// TwinCAT 3 PLC project TcLog
// Title: TcLog
// Company: TcLog
// ProjectVersion: 0.5.0
// ProgramVersion: 3.1.4022.7
// libraries:
//   Tc2_Standard, * (Beckhoff Automation GmbH)
//   Tc2_System, * (Beckhoff Automation GmbH)
//   Tc2_Utilities, * (Beckhoff Automation GmbH)
//   Tc3_Module, * (Beckhoff Automation GmbH)
//   TcExt, * (TcExt)
//   TcUnit, * (www.tcunit.org)
// project tree:
//   Event/ CyclicEventDetection.TcPOU, EventMessageHMI.TcDUT, ST_CyclicMessageDetection.TcDUT, Event.TcPOU, EventLevel.TcDUT, EventMessage.TcDUT, EventRunner.TcPOU, ST_CyclicEventDetection.TcDUT
//   / GlobalTextList.TcGTLO, SymbolsPool.TcIPO (not stored), Visualization Manager.TcVMO (not stored)
//   GVL/ GVL.TcGVL, Properties.TcGVL
//   Logger/ ADSLogger.TcPOU, EventLogger.TcIO, CSVLogger.TcPOU, MemoryLogger.TcPOU, AlarmViewLogger.TcPOU
//   Tests/Event/ EventTestsystem.TcDUT, MultipleEventTestsystem.TcDUT, TestEvent.TcPOU
//   Tests/Logger/ ADSLoggerTestsystem.TcDUT, CSVLoggerTestsystem.TcDUT, TestADSLogger.TcPOU, TestCSVLogger.TcPOU
//   Tests/ PlcTask.TcTTO, TEST_MAIN.TcPOU, TEST_STRING_CYCLE_TIME.TcPOU
//   Tests/Utils/ TestUtils.TcPOU
//   Utils/ FB_FrameFifo.TcPOU, LString.TcPOU, put_new_data_at_start.TcPOU, remove_field_from_array.TcPOU, TIMESTRUCT_TO_DATESTR.TcPOU, TIMESTRUCT_TO_TIMESTR.TcPOU, TO_LSTRING.TcPOU
//   Visu/ AlarmViewMulti.TcVIS, AlarmViewSingle.TcVIS, AlarmViewSingleWithReset.TcVIS
// real-time tasks:
//   TASK PlcTask: cycle T#10ms, priority 20, ADS port 350

CONFIGURATION TcLog
    RESOURCE PLC ON TwinCAT3
        TASK PlcTask(INTERVAL := T#10ms, PRIORITY := 20);
    END_RESOURCE
END_CONFIGURATION

// ---- Event/EventMessageHMI.TcDUT
TYPE EventMessageHMI :
STRUCT
  id: INT;
  timestamp: STRING;
  path: STRING;
  message: STRING;
  level: EventLevel;
END_STRUCT
END_TYPE

// ---- Event/ST_CyclicMessageDetection.TcDUT
TYPE ST_CyclicMessageDetection :
STRUCT
  ev: EventMessage;
  message_submitted: BOOL;
END_STRUCT
END_TYPE

// ---- Event/EventLevel.TcDUT
{attribute 'qualified_only'}
{attribute 'strict'}
{attribute 'to_string'}
TYPE EventLevel :
(
  NONE := 0,
  DEBUG := 1,
	INFO := 2,
  WARNING := 3,
  ERROR := 4,
  ALARM := 5
) BYTE := NONE;
END_TYPE

// ---- Event/EventMessage.TcDUT
TYPE EventMessage :
STRUCT
  id: INT;
  path: LString;
  message: LString;
  level: EventLevel;
  cleared: BOOL;
END_STRUCT
END_TYPE

// ---- Event/ST_CyclicEventDetection.TcDUT
TYPE ST_CyclicEventDetection :
STRUCT
  id: INT;
  submitted_in_last_invocation: BIT;
END_STRUCT
END_TYPE

// ---- Tests/Event/EventTestsystem.TcDUT
TYPE EventTestsystem :
STRUCT
  logging: EventRunner;
  event: Event := (logging:=logging);
END_STRUCT
END_TYPE

// ---- Tests/Event/MultipleEventTestsystem.TcDUT
TYPE MultipleEventTestsystem :
STRUCT
  logging: EventRunner;
  event1: Event := (logging:=logging);
  event2: Event := (logging:=logging);
  event3: Event := (logging:=logging);
END_STRUCT
END_TYPE

// ---- Tests/Logger/ADSLoggerTestsystem.TcDUT
TYPE ADSLoggerTestsystem :
STRUCT
  logging: EventRunner;
  event: Event := (logging:=logging);
  logger: ADSLogger := (disable_ads_output := TRUE);
END_STRUCT
END_TYPE

// ---- Tests/Logger/CSVLoggerTestsystem.TcDUT
TYPE CSVLoggerTestsystem :
STRUCT
  logging: EventRunner;
  event: Event := (logging:=logging);
  logger: CSVLogger;
END_STRUCT
END_TYPE

// ---- GVL/GVL.TcGVL
VAR_GLOBAL
  logging: EventRunner;
END_VAR
VAR_GLOBAL CONSTANT
  EXCLUDE_ID: INT := 0;
  // Index zero should not be visible
  IMAGE_ID: ARRAY[0..5] OF STRING(20) := ['SymbolsPool.info', 'SymbolsPool.info', 'SymbolsPool.info', 'SymbolsPool.warning', 'SymbolsPool.error', 'SymbolsPool.alarm'];
END_VAR

// ---- GVL/Properties.TcGVL
{attribute 'qualified_only'}
VAR_GLOBAL CONSTANT
  NUM_EVENTS: INT := 500;
  NUM_CONCURRENT_ALARMS: INT := 10;
  NUM_LOGGER: INT := 5;
  NUM_CYCLIC_DETECTION_MESSAGES: INT := 10;
  CSV_BUFFER_SIZE: UDINT := 2000;
  MEMORY_LOGGER_NUM_EVENTS_HISTORY: INT := 100;
  MEMORY_LOGGER_NUM_EVENTS_HMI: INT := 30;
  ALARM_VIEW_NUM_EVENTS: INT := 20;
END_VAR

// ---- Logger/EventLogger.TcIO
INTERFACE EventLogger

METHOD clear_event_message
VAR_INPUT
  id: INT;
END_VAR
END_METHOD

PROPERTY PUBLIC level : EventLevel
GET
END_GET
SET
END_SET
END_PROPERTY

METHOD run
VAR_INPUT
  act_time: TIMESTRUCT;
END_VAR
END_METHOD

METHOD PUBLIC submit_event_message
VAR_IN_OUT
  ev: EventMessage;
END_VAR
END_METHOD

END_INTERFACE

// ---- Event/EventRunner.TcPOU
{attribute 'reflection'}
FUNCTION_BLOCK EventRunner
VAR_INPUT
END_VAR
VAR_OUTPUT
END_VAR
VAR
  {attribute 'instance-path'}
  {attribute 'noinit'}
  path_str: STRING(255);
  path: LString;
  event_id_counter: INT;
  localtime: FB_LocalSystemTime := (bEnable:=TRUE);
  actSystemTime: TIMESTRUCT;
  event_logger: ARRAY[1..Properties.NUM_LOGGER] OF EventLogger;
  active_alarms: ARRAY[1..Properties.NUM_CONCURRENT_ALARMS] OF EventMessage;
  detection: CyclicEventDetection;
  logger_counter: INT;
  format_str: FB_FormatString;
  _parameter: T_Arg;
  
  submit_event_message_counter: INT;
  max_submit_event_message_counter: INT;
END_VAR

(* 
der runner wird am ende des sps programms ausgefuehrt
- im programm werden pro meldung event-instanzen erstellt. diese registrieren sich selbst. die richtige id wird der pfad zur instanzvariable sein
- im runner wird zudem das datum immer aktualisiert
*)

PROPERTY PRIVATE act_time : TIMESTRUCT
GET
IF time_valid THEN
  act_time := localtime.systemTime;
END_IF
END_GET
END_PROPERTY

METHOD PUBLIC add_logger
VAR_INPUT
  logger: EventLogger;
END_VAR
IF logger_counter < Properties.NUM_LOGGER AND ADR(logger) <> 0 AND NOT logger_exist(logger) THEN
  inc_logger_counter();
  event_logger[logger_counter] := logger;
END_IF
END_METHOD

METHOD INTERNAL alarm_raised : BOOL
VAR_INPUT
  id: INT;
END_VAR
VAR
  i: INT;
END_VAR
alarm_raised := get_alarm_index(id:=id) > 0;
END_METHOD

METHOD PUBLIC clear
VAR_INPUT
  id: INT;
END_VAR
VAR
  i: INT;
END_VAR
FOR i:=1 TO Properties.NUM_LOGGER DO
  IF event_logger[i] <> 0 THEN
    event_logger[i].clear_event_message(id);
	END_IF
END_FOR
END_METHOD

METHOD INTERNAL clear_alarm
VAR_INPUT
  id: INT;
END_VAR
VAR
  index: INT;
  filldata: EventMessage;
END_VAR
IF alarm_raised(id:=id) THEN
  index := get_alarm_index(id:=id);
  active_alarms[index].cleared := TRUE;
  
  submit_event_message_to_logger(active_alarms[index]);
  
  remove_field_from_array(
    index_to_remove:=index,
    size_filldata:=SIZEOF(filldata),
    adr_filldata:=ADR(filldata),
    size_memory_buffer:=SIZEOF(active_alarms),
    adr_memory_buffer:=ADR(active_alarms));
END_IF
END_METHOD

METHOD PRIVATE create_event_message
VAR_INPUT
  id: INT;
  level: EventLevel;
  cleared: BOOL;
END_VAR
VAR_IN_OUT
  ev: EventMessage;
  path: LString;
  message: LString;
END_VAR
VAR
  undefined_time: TIMESTRUCT;
  num_dots: INT;
  i: INT;
  offset: INT;
END_VAR
ev.id := id;
ev.path := path;
ev.message := message;
ev.level := level;
ev.cleared := cleared;
END_METHOD

METHOD PUBLIC error
VAR_INPUT
  message: STRING(255);
END_VAR
VAR_INST
  message_lstr: LString;
END_VAR
message_lstr := TO_LSTRING(message);
submit_message(
  message:=message_lstr,
  level:=EventLevel.ERROR);
END_METHOD

METHOD PUBLIC error_if_true
VAR_INPUT
  value: BOOL;
  message: STRING(255);
END_VAR
IF value THEN
  error(message);
END_IF
END_METHOD

METHOD FB_init : BOOL
VAR_INPUT
	bInitRetains : BOOL; // if TRUE, the retain variables are initialized (warm start / cold start)
	bInCopyCode : BOOL;  // if TRUE, the instance afterwards gets moved into the copy code (online change)
END_VAR
path.str := path_str;
END_METHOD

METHOD INTERNAL generate_event_id : INT
VAR_INPUT
END_VAR
inc_event_id_counter();
generate_event_id := event_id_counter;
END_METHOD

METHOD PRIVATE get_alarm_index : INT
VAR_INPUT
  id: INT;
END_VAR
VAR
  i: INT;
END_VAR
get_alarm_index := 0;
FOR i:=1 TO Properties.NUM_CONCURRENT_ALARMS DO
  IF active_alarms[i].id = id AND NOT active_alarms[i].cleared THEN
    get_alarm_index := i;
    EXIT;
	END_IF
END_FOR
END_METHOD

METHOD PRIVATE inc_event_id_counter
VAR_INPUT
END_VAR
event_id_counter := LIMIT(1, event_id_counter + 1, Properties.NUM_EVENTS);
END_METHOD

METHOD PRIVATE inc_logger_counter
VAR_INPUT
END_VAR
logger_counter := LIMIT(1, logger_counter + 1, Properties.NUM_LOGGER);
END_METHOD

METHOD PUBLIC info
VAR_INPUT
  message: STRING(255);
END_VAR
VAR_INST
  message_lstr: LString;
END_VAR
message_lstr := TO_LSTRING(message);
submit_message(
  message:=message_lstr,
  level:=EventLevel.INFO);
END_METHOD

METHOD PUBLIC info_if_true
VAR_INPUT
  value: BOOL;
  message: STRING(255);
END_VAR
IF value THEN
  info(message);
END_IF
END_METHOD

METHOD PRIVATE logger_exist : BOOL
VAR_INPUT
  logger: EventLogger;
END_VAR
VAR
  i: INT;
END_VAR
logger_exist := FALSE;
FOR i:=1 TO Properties.NUM_LOGGER DO
  IF event_logger[i] = logger THEN
    logger_exist := TRUE;
    EXIT;
	END_IF
END_FOR
END_METHOD

PROPERTY PUBLIC parameter : T_Arg
GET
parameter := _parameter;
END_GET
SET
_parameter := parameter;
END_SET
END_PROPERTY

METHOD PUBLIC reset_events_and_messages
VAR_INPUT
END_VAR
detection.reset_events();
detection.reset_messages();
END_METHOD

METHOD PUBLIC run
VAR_INPUT
END_VAR
VAR
  read_done: BOOL;
  error_id: UDINT;
END_VAR
localtime();
run_logger();
detection.cyclic_call();
submit_event_message_counter := 0;
END_METHOD

METHOD PRIVATE run_logger
VAR_INPUT
END_VAR
VAR
  i: INT;
END_VAR
FOR i:=1 TO Properties.NUM_LOGGER DO
  IF event_logger[i] <> 0 THEN
    event_logger[i].run(act_time:=act_time);
	END_IF
END_FOR
END_METHOD

METHOD PUBLIC submit_event
VAR_INPUT
  id: INT;
  level: EventLevel;
  cleared: BOOL;
END_VAR
VAR_IN_OUT
  path: LString;
  message: LString;
END_VAR
VAR
  temp_message: STRING(255);
END_VAR
VAR_INST
  ev: EventMessage;
  event_index: INT;
  message_index: INT;
  formatted_message: LString;
END_VAR
IF alarm_raised(id:=id) THEN
  RETURN;
END_IF

event_index := detection.get_event_index(id);
IF event_index = 0 THEN
  detection.add_event(id);
  IF _parameter.cbLen > 0 THEN
    format_str(
      sFormat:=message.str,
      arg1:=parameter,
      sOut=>temp_message);
    formatted_message.str := temp_message;
  ELSE
    formatted_message := message;
  END_IF
  ev.id := id;
  ev.path := path;
  ev.message := formatted_message;
  ev.level := level;
  ev.cleared := cleared;
  ev.path.remove_left_including_char('.', 2);
  submit_event_message_to_logger(ev);
  
  IF NOT cleared THEN
    put_new_data_at_start(SIZEOF(ev), ADR(ev), SIZEOF(active_alarms), ADR(active_alarms));
  END_IF
ELSE
  detection.reactivate_event(event_index);
END_IF
END_METHOD

METHOD PRIVATE submit_event_message_to_logger
VAR_IN_OUT
  ev: EventMessage;
END_VAR
VAR
  i: INT;
END_VAR
FOR i:=1 TO Properties.NUM_LOGGER DO
  IF event_logger[i] <> 0 THEN
    event_logger[i].submit_event_message(ev);
	END_IF
END_FOR
END_METHOD

METHOD PRIVATE submit_message
VAR_INPUT
  level: EventLevel;
END_VAR
VAR_IN_OUT
  message: LString;
END_VAR
VAR
  temp_message: STRING(255);
END_VAR
VAR_INST
  ev: EventMessage;
  event_index: INT;
  message_index: INT;
  formatted_message: LString;
END_VAR
IF _parameter.cbLen > 0 THEN
  format_str(
    sFormat:=message.str,
    arg1:=parameter,
    sOut=>temp_message);
  formatted_message.str := temp_message;
ELSE
  formatted_message := message;
END_IF
create_event_message(
    ev:=ev,
    id:=GVL.EXCLUDE_ID,
    path:=path,
    message:=formatted_message,
    level:=level,
    cleared:=TRUE);
message_index := detection.get_message_index(ev);
IF message_index = 0 THEN
  ev.path.remove_left_including_char('.', 2);
  detection.add_message(ev);
  
  submit_event_message_to_logger(ev);
ELSE
  detection.reactivate_message(message_index);
END_IF
END_METHOD

PROPERTY PUBLIC time_valid : BOOL
GET
time_valid := localtime.bValid;
END_GET
END_PROPERTY

METHOD PRIVATE timestruct_equal : BOOL
VAR_INPUT
  timestruct_1: TIMESTRUCT;
  timestruct_2: TIMESTRUCT;
END_VAR
timestruct_equal := timestruct_1.wDay = timestruct_2.wDay;
timestruct_equal := timestruct_equal AND timestruct_1.wDayOfWeek = timestruct_2.wDayOfWeek;
timestruct_equal := timestruct_equal AND timestruct_1.wHour = timestruct_2.wHour;
timestruct_equal := timestruct_equal AND timestruct_1.wMilliseconds = timestruct_2.wMilliseconds;
timestruct_equal := timestruct_equal AND timestruct_1.wMinute = timestruct_2.wMinute;
END_METHOD

METHOD PUBLIC warning
VAR_INPUT
  message: STRING(255);
END_VAR
VAR_INST
  message_lstr: LString;
END_VAR
message_lstr := TO_LSTRING(message);
submit_message(
  message:=message_lstr,
  level:=EventLevel.WARNING);
END_METHOD

METHOD PUBLIC warning_if_true
VAR_INPUT
  value: BOOL;
  message: STRING(255);
END_VAR
IF value THEN
  warning(message);
END_IF
END_METHOD

END_FUNCTION_BLOCK

// ---- Utils/LString.TcPOU
FUNCTION_BLOCK LString
VAR_INPUT
END_VAR
VAR_OUTPUT
END_VAR
VAR
  _str: STRING(255);
  _length: INT;
END_VAR

METHOD PUBLIC append
VAR_IN_OUT
  lstr: LString; 
END_VAR
MEMMOVE(
  destAddr:=ADR(_str)+TO_DWORD(length),
  srcAddr:=ADR(lstr._str),
  n:=TO_UDINT(lstr.length+1));
length := length + lstr.length;
END_METHOD

METHOD PUBLIC append_str
VAR_INPUT
  str: STRING(255);
END_VAR
VAR
  length: INT;
END_VAR
length := LEN(str);
MEMMOVE(
  destAddr:=ADR(_str)+TO_DWORD(THIS^.length),
  srcAddr:=ADR(str),
  n:=TO_UDINT(length+1));
THIS^.length := THIS^.length + length;
END_METHOD

PROPERTY PUBLIC length : INT
GET
length := _length;
END_GET
SET // PRIVATE
_length := length;
END_SET
END_PROPERTY

METHOD PUBLIC remove_left_including_char
VAR_INPUT
  char: STRING(1);
  number: INT;
END_VAR
VAR
  act_number: INT;
  offset: INT;
  i: INT;
END_VAR
WHILE _str[i] <> 0 DO
  IF act_number < number THEN
    IF _str[i] = char[0] THEN
      act_number := act_number + 1;
    END_IF
  ELSE
    EXIT;
	END_IF
  i := i + 1;
END_WHILE
MEMMOVE(
  destAddr:=ADR(_str),
  srcAddr:=ADR(_str)+TO_DWORD(i),
  n:=TO_UDINT(length-i));
length := length - i;
_str[length] := 0;
END_METHOD

PROPERTY PUBLIC str : STRING(255)
GET
str := _str;
END_GET
SET
_str := str;
length := LEN(str);
END_SET
END_PROPERTY

END_FUNCTION_BLOCK

// ---- Event/CyclicEventDetection.TcPOU
FUNCTION_BLOCK CyclicEventDetection
VAR_INPUT
END_VAR
VAR_OUTPUT
END_VAR
VAR
  message_counter: INT;
  event_counter: INT;
  messages: ARRAY[1..Properties.NUM_CYCLIC_DETECTION_MESSAGES] OF ST_CyclicMessageDetection;
  events: ARRAY[1..Properties.NUM_EVENTS] OF ST_CyclicEventDetection;
END_VAR

METHOD PRIVATE activate_event
VAR_INPUT
  index: INT;
END_VAR
events[index].submitted_in_last_invocation := TRUE;
END_METHOD

METHOD PRIVATE activate_message
VAR_INPUT
  index: INT;
END_VAR
messages[index].message_submitted := TRUE;
END_METHOD

METHOD PUBLIC add_event
VAR_INPUT
  id: INT;
END_VAR
VAR
  event_index: INT;
END_VAR
inc_event_counter();
events[event_counter].id := id;
activate_event(event_counter);
END_METHOD

METHOD PUBLIC add_message
VAR_INPUT
  ev: EventMessage;
END_VAR
VAR
  event_index: INT;
END_VAR
IF NOT max_number_events_reached() THEN
  inc_message_counter();
  messages[message_counter].ev := ev;
  activate_message(message_counter);
END_IF
END_METHOD

METHOD PUBLIC cyclic_call
VAR_INPUT
END_VAR
remove_deactivated_events();
remove_deactivated_messages();
reset_events();
reset_messages();
END_METHOD

METHOD PRIVATE dec_event_counter
VAR_INPUT
END_VAR
event_counter := LIMIT(0, event_counter - 1, Properties.NUM_EVENTS);
END_METHOD

METHOD PRIVATE dec_message_counter
VAR_INPUT
END_VAR
message_counter := LIMIT(0, message_counter - 1, Properties.NUM_CYCLIC_DETECTION_MESSAGES);
END_METHOD

METHOD PRIVATE event_id_valid : BOOL
VAR_INPUT
  id: INT;
END_VAR
event_id_valid := (1 <= id) AND (id <= Properties.NUM_EVENTS);
END_METHOD

METHOD PUBLIC event_was_called_in_last_invocation : BOOL
VAR_INPUT
  id: INT;
END_VAR
VAR
  i: INT;
END_VAR
FOR i:=1 TO event_counter DO
  IF events[i].id = id THEN
    event_was_called_in_last_invocation := TRUE;
    EXIT;
	END_IF
END_FOR
END_METHOD

METHOD PUBLIC get_event_index : INT
VAR_INPUT
  id: INT;
END_VAR
VAR
  i: INT;
END_VAR
FOR i:=1 TO event_counter DO
  IF events[i].id = id THEN
    get_event_index := i;
    EXIT;
  END_IF
END_FOR
END_METHOD

METHOD get_message_index : INT
VAR_IN_OUT
  ev: EventMessage;
END_VAR
VAR
  i: INT;
END_VAR
FOR i:=1 TO message_counter DO
  IF messages[i].ev.message.str = ev.message.str THEN
    get_message_index := i;
    EXIT;
  END_IF
END_FOR
END_METHOD

METHOD PRIVATE inc_event_counter
VAR_INPUT
END_VAR
event_counter := LIMIT(1, event_counter + 1, Properties.NUM_EVENTS);
END_METHOD

METHOD PRIVATE inc_message_counter
VAR_INPUT
END_VAR
message_counter := LIMIT(1, message_counter + 1, Properties.NUM_CYCLIC_DETECTION_MESSAGES);
END_METHOD

METHOD PRIVATE max_number_events_reached : BOOL
VAR_INPUT
END_VAR
max_number_events_reached := message_counter >= Properties.NUM_CYCLIC_DETECTION_MESSAGES;
END_METHOD

METHOD PRIVATE message_index_valid : BOOL
VAR_INPUT
  index: INT;
END_VAR
message_index_valid := (1 <= index) AND (index <= Properties.NUM_CYCLIC_DETECTION_MESSAGES);
END_METHOD

METHOD PUBLIC reactivate_event
VAR_INPUT
  index: INT;
END_VAR
IF event_id_valid(index) THEN
  activate_event(index);
END_IF
END_METHOD

METHOD PUBLIC reactivate_message
VAR_INPUT
  index: INT;
END_VAR
IF event_id_valid(index) THEN
  activate_message(index);
END_IF
END_METHOD

METHOD PRIVATE remove_deactivated_events
VAR_INPUT
END_VAR
VAR
  i: INT;
  filldata: ST_CyclicEventDetection;
END_VAR
FOR i:=1 TO event_counter DO
  IF NOT events[i].submitted_in_last_invocation THEN
    remove_field_from_array(
      index_to_remove:=i,
      size_filldata:=SIZEOF(filldata),
      adr_filldata:=ADR(filldata),
      size_memory_buffer:=SIZEOF(events),
      adr_memory_buffer:=ADR(events)
    );
    dec_event_counter();
    i := i - 1;
	END_IF
END_FOR
END_METHOD

METHOD PRIVATE remove_deactivated_messages
VAR_INPUT
END_VAR
VAR
  i: INT;
  filldata: ST_CyclicMessageDetection;
END_VAR
FOR i:=1 TO message_counter DO
  IF NOT messages[i].message_submitted THEN
    remove_field_from_array(
      index_to_remove:=i,
      size_filldata:=SIZEOF(filldata),
      adr_filldata:=ADR(filldata),
      size_memory_buffer:=SIZEOF(messages),
      adr_memory_buffer:=ADR(messages)
    );
    dec_message_counter();
    i := i - 1;
	END_IF
END_FOR
END_METHOD

METHOD PRIVATE reset_event
VAR_INPUT
  index: INT;
END_VAR
events[index].submitted_in_last_invocation := FALSE;
END_METHOD

METHOD PUBLIC reset_events
VAR_INPUT
END_VAR
VAR
  i: INT;
END_VAR
FOR i:=1 TO event_counter DO
  reset_event(i);
END_FOR
END_METHOD

METHOD PRIVATE reset_message
VAR_INPUT
  index: INT;
END_VAR
messages[index].message_submitted := FALSE;
END_METHOD

METHOD PUBLIC reset_messages
VAR_INPUT
END_VAR
VAR
  i: INT;
END_VAR
FOR i:=1 TO message_counter DO
  reset_message(i);
END_FOR
END_METHOD

END_FUNCTION_BLOCK

// ---- Utils/remove_field_from_array.TcPOU
FUNCTION remove_field_from_array : BOOL
VAR_INPUT
  index_to_remove: INT; // array index must start with 1
  size_filldata: UDINT;
  adr_filldata: POINTER TO BYTE; 
  size_memory_buffer: UDINT;
  adr_memory_buffer : POINTER TO BYTE;
END_VAR
VAR
END_VAR

IF index_to_remove < 1 THEN
  RETURN;
END_IF

(*
example:
size_memory_buffer = 20
size_filldata = 1
index_to_remove = 1
adr_memory_buffer = 100
---------------------------------
size_new_data = 20 - 1 = 19
adr_new_data = 100 + 1 = 101


size_memory_buffer = 20 - 1 = 19
adr_memory_buffer = 100 + 0 = 100
*)

FW_MemMove(
  pDest := adr_memory_buffer + size_filldata*TO_UDINT((index_to_remove-1)),
  pSrc := adr_memory_buffer + size_filldata*TO_UDINT(index_to_remove),
  cbLen := size_memory_buffer - size_filldata*TO_UDINT(index_to_remove));
FW_MemMove(
  pDest := adr_memory_buffer + (size_memory_buffer - size_filldata),
  pSrc := adr_filldata,
  cbLen := size_filldata);

END_FUNCTION

// ---- Utils/TO_LSTRING.TcPOU
FUNCTION TO_LSTRING : LSTRING
VAR_INPUT
  str: STRING(255);
END_VAR
VAR
END_VAR

TO_LSTRING.str := str;

END_FUNCTION

// ---- Utils/put_new_data_at_start.TcPOU
FUNCTION put_new_data_at_start: BOOL
VAR_INPUT
  size_new_data: UDINT;
  adr_new_data: POINTER TO BYTE;

  size_memory_buffer: UDINT;
  adr_memory_buffer : POINTER TO BYTE;
END_VAR

FW_MemMove(
  pDest := adr_memory_buffer + size_new_data,
  pSrc := adr_memory_buffer,
  cbLen := size_memory_buffer - size_new_data);
FW_MemMove(
  pDest := adr_memory_buffer,
  pSrc := adr_new_data,
  cbLen := size_new_data);

END_FUNCTION

// ---- Event/Event.TcPOU
{attribute 'reflection'}
FUNCTION_BLOCK Event
VAR_INPUT
END_VAR
VAR_OUTPUT
END_VAR
VAR
  _logging: REFERENCE TO EventRunner;
  {attribute 'instance-path'}
  {attribute 'noinit'}
  path_str: STRING(255);
  path: LString;
  id: INT;
  _message: LString;
  _parameter: T_Arg;
  ev: EventMessage;
END_VAR

METHOD PUBLIC alarm
VAR_INPUT
END_VAR
submit(level:=EventLevel.ALARM);
END_METHOD

METHOD alarm_if_true
VAR_INPUT
    value: BOOL;
END_VAR
IF value THEN
  alarm();
ELSE
  clear_alarm();
END_IF
END_METHOD

PROPERTY PUBLIC alarm_raised : BOOL
GET
alarm_raised := logging.alarm_raised(id);
END_GET
END_PROPERTY

METHOD PUBLIC clear
VAR_INPUT
END_VAR
logging.clear(id:=id);
END_METHOD

METHOD PUBLIC clear_alarm
VAR_INPUT
END_VAR
logging.clear_alarm(id:=id);
END_METHOD

METHOD PUBLIC debug
VAR_INPUT
END_VAR
submit(level:=EventLevel.DEBUG);
END_METHOD

METHOD debug_if_true
VAR_INPUT
  value: BOOL;
END_VAR
VAR_INST
  r_value: R_TRIG;
END_VAR
r_value(CLK:=value);
IF r_value.Q THEN
  debug();
END_IF
END_METHOD

METHOD debug_signal
VAR_INPUT
  signal: BOOL;
END_VAR
IF signal THEN
  debug();
ELSE
  clear();
END_IF
END_METHOD

METHOD PUBLIC error
VAR_INPUT
END_VAR
submit(level:=EventLevel.ERROR);
END_METHOD

METHOD error_if_true
VAR_INPUT
  value: BOOL;
END_VAR
VAR_INST
  r_value: R_TRIG;
END_VAR
r_value(CLK:=value);
IF r_value.Q THEN
  error();
END_IF
END_METHOD

METHOD error_signal
VAR_INPUT
  signal: BOOL;
END_VAR
IF signal THEN
  error();
ELSE
  clear();
END_IF
END_METHOD

METHOD FB_init : BOOL
VAR_INPUT
	bInitRetains : BOOL; // if TRUE, the retain variables are initialized (warm start / cold start)
	bInCopyCode : BOOL;  // if TRUE, the instance afterwards gets moved into the copy code (online change)
END_VAR
THIS^.logging REF= GVL.logging;
path.str := path_str;
END_METHOD

METHOD info
VAR_INPUT
END_VAR
submit(level:=EventLevel.INFO);
END_METHOD

METHOD info_if_true
VAR_INPUT
  value: BOOL;
END_VAR
VAR_INST
  r_value: R_TRIG;
END_VAR
r_value(CLK:=value);
IF r_value.Q THEN
  info();
END_IF
END_METHOD

PROPERTY PUBLIC logging : REFERENCE TO EventRunner
GET
logging REF= _logging;
END_GET
SET
_logging REF= logging;
set_id(logging.generate_event_id());
END_SET
END_PROPERTY

PROPERTY PUBLIC message : STRING(255)
GET
message := _message.str;
END_GET
SET
_message.str := message;
END_SET
END_PROPERTY

PROPERTY PUBLIC parameter : T_Arg
GET
parameter := _parameter;
END_GET
SET
_parameter := parameter;
END_SET
END_PROPERTY

METHOD PRIVATE set_id
VAR_INPUT
  id: INT;
END_VAR
THIS^.id := id;
END_METHOD

METHOD PRIVATE submit
VAR_INPUT
  level: EventLevel;
END_VAR
logging.parameter := parameter;
logging.submit_event(
  id:=id,
  path:=path,
  message:=_message,
  level:=level,
  cleared:=level <> EventLevel.ALARM);
END_METHOD

METHOD warning
VAR_INPUT
END_VAR
submit(level:=EventLevel.WARNING);
END_METHOD

METHOD warning_if_true
VAR_INPUT
  value: BOOL;
END_VAR
VAR_INST
  r_value: R_TRIG;
END_VAR
r_value(CLK:=value);
IF r_value.Q THEN
  warning();
END_IF
END_METHOD

METHOD warning_signal
VAR_INPUT
  signal: BOOL;
END_VAR
IF signal THEN
  warning();
ELSE
  clear();
END_IF
END_METHOD

END_FUNCTION_BLOCK

// ---- Logger/ADSLogger.TcPOU
FUNCTION_BLOCK ADSLogger IMPLEMENTS EventLogger
VAR_INPUT
END_VAR
VAR_OUTPUT
END_VAR
VAR
  _level: EventLevel;
  _disable_ads_output: BOOL;
  _mask: DWORD;
  _ref_formatted_output: REFERENCE TO LString;
  _formatted_output: LString;
  _path: STRING(255);
END_VAR

METHOD PRIVATE ads_log
VAR_IN_OUT
  ev: EventMessage;
END_VAR
VAR
END_VAR
mask := create_mask(ev.level);

formatted_output := ev.path;
formatted_output.append_str(' | ');
formatted_output.append_str(TO_STRING(ev.level));
formatted_output.append_str(': ');
formatted_output.append(ev.message);

IF NOT disable_ads_output THEN
  ADSLOGSTR(mask, formatted_output.str, '');
END_IF
END_METHOD

METHOD clear_event_message
VAR_INPUT
	id: INT;
END_VAR
// nothing to do here
END_METHOD

METHOD PRIVATE create_mask : DWORD
VAR_IN_OUT
  level: EventLevel;
END_VAR
CASE level OF
EventLevel.INFO:
  create_mask := ADSLOG_MSGTYPE_HINT;
EventLevel.WARNING:
  create_mask := ADSLOG_MSGTYPE_WARN;
EventLevel.ERROR, EventLevel.ALARM:
  create_mask := ADSLOG_MSGTYPE_ERROR;
ELSE
  create_mask := ADSLOG_MSGTYPE_HINT;
END_CASE
END_METHOD

PROPERTY INTERNAL disable_ads_output : BOOL
GET
disable_ads_output := _disable_ads_output;
END_GET
SET
_disable_ads_output := disable_ads_output;
END_SET
END_PROPERTY

METHOD FB_init : BOOL
VAR_INPUT
	bInitRetains : BOOL; // if TRUE, the retain variables are initialized (warm start / cold start)
	bInCopyCode : BOOL;  // if TRUE, the instance afterwards gets moved into the copy code (online change)
END_VAR
formatted_output REF= _formatted_output;
END_METHOD

PROPERTY INTERNAL formatted_output : REFERENCE TO LString
GET
formatted_output REF= _ref_formatted_output;
END_GET
SET // PRIVATE
_ref_formatted_output REF= formatted_output;
END_SET
END_PROPERTY

PROPERTY PUBLIC level : EventLevel
GET
level := _level;
END_GET
SET
_level := level;
END_SET
END_PROPERTY

PROPERTY INTERNAL mask : DWORD
GET
mask := _mask;
END_GET
SET // PRIVATE
_mask := mask;
END_SET
END_PROPERTY

PROPERTY INTERNAL path : STRING(255)
GET
path := _path;
END_GET
SET // PRIVATE
_path := path;
END_SET
END_PROPERTY

METHOD run
VAR_INPUT
  act_time: TIMESTRUCT;
END_VAR
(* 
nothing to do here. a proposal would be to implement a buffered
approach like TcUnit did in issue #35 because too many ADSLOGSTR
calls could lead to a loss of messages.
*)
;
END_METHOD

METHOD PUBLIC submit_event_message
VAR_IN_OUT
	ev: EventMessage;
END_VAR
IF ev.level >= level THEN
  ads_log(ev);
END_IF
END_METHOD

END_FUNCTION_BLOCK

// ---- Logger/CSVLogger.TcPOU
FUNCTION_BLOCK CSVLogger IMPLEMENTS EventLogger
VAR_INPUT
END_VAR
VAR_OUTPUT
END_VAR
VAR
  _path: STRING(255);
  filename: STRING(255);
  file: TcExt.FileMemory := (mode_write := Tc2_System.FOPEN_MODEAPPEND OR Tc2_System.FOPEN_MODETEXT);
  _done: BOOL;
  _level: EventLevel;
  act_time: TIMESTRUCT;
  act_time_str: STRING(255);
  _datetime_format: STRING(255) := '%4.0f-%02.0f-%02.0f %02.0f:%02.0f:%02.0f.%03.0f';
  format_string: FB_FormatString;
  message_queue: FB_FrameFifo;
  state_number: INT;
  formatted_output: LString;
END_VAR

METHOD clear_event_message
VAR_INPUT
	id: INT;
END_VAR
// nothing to do here
END_METHOD

METHOD INTERNAL create_row
VAR_IN_OUT
  ev: EventMessage;
END_VAR
VAR
END_VAR
formatted_output := TO_LSTRING(act_time_str);
formatted_output.append_str(',');
formatted_output.append_str(TO_STRING(ev.cleared));
formatted_output.append_str(',');
formatted_output.append_str(TO_STRING(ev.level));
formatted_output.append_str(',');
formatted_output.append(ev.path);
formatted_output.append_str(',');
formatted_output.append(ev.message);
formatted_output.append_str('$R');
END_METHOD

PROPERTY PUBLIC datetime_format : STRING(255)
GET
datetime_format := _datetime_format;
END_GET
SET
_datetime_format := datetime_format;
END_SET
END_PROPERTY

METHOD PRIVATE get_timestamped_filename
VAR_IN_OUT
  filename: STRING(255);
END_VAR
TIMESTRUCT_TO_DATESTR(
  ts:=act_time,
  outputstr:=filename);
format_string(
  sFormat:='log_%s.csv',
  arg1:=F_STRING(filename),
  sOut=>filename);
END_METHOD

PROPERTY PUBLIC level : EventLevel
GET
level := _level;
END_GET
SET
_level := level;
END_SET
END_PROPERTY

PROPERTY PUBLIC path : STRING(255)
GET
path := _path;
END_GET
SET
_path := path;
END_SET
END_PROPERTY

METHOD run
VAR_INPUT
  act_time: TIMESTRUCT;
END_VAR
VAR_INST
  year: REAL;
  month: REAL;
  day: REAL;
  hour: REAL;
  minute: REAL;
  second: REAL;
  millisecond: REAL;
END_VAR
THIS^.act_time := act_time;
// ugly hack. have to convert numbers to real because the format specification
// only allows leading zeros on types f, e and s
year := TO_REAL(act_time.wYear);
month := TO_REAL(act_time.wMonth);
day := TO_REAL(act_time.wDay);
hour := TO_REAL(act_time.wHour);
minute := TO_REAL(act_time.wMinute);
second := TO_REAL(act_time.wSecond);
millisecond := TO_REAL(act_time.wMilliseconds);
format_string(
  sFormat:=datetime_format,
  arg1:=F_REAL(year),
  arg2:=F_REAL(month),
  arg3:=F_REAL(day),
  arg4:=F_REAL(hour),
  arg5:=F_REAL(minute),
  arg6:=F_REAL(second),
  arg7:=F_REAL(millisecond),
  sOut=>act_time_str);

save();
END_METHOD

METHOD PRIVATE save
VAR
  done: BOOL;
  error_id: DWORD;
  
END_VAR
CASE state_number OF
0:
  message_queue.RemoveHead();
  IF message_queue.bOk THEN
    get_timestamped_filename(filename);
    file.path := CONCAT(path, filename);
    file.write(
      start:=FALSE,
      data_ptr:=ADR(message_queue.sGet),
      data_size:=TO_UDINT(LEN(message_queue.sGet))
    );
    state_number := state_number + 10;
	END_IF
10:
  file.write(
    start:=TRUE,
    data_ptr:=ADR(message_queue.sGet),
    data_size:=TO_UDINT(LEN(message_queue.sGet)),
    done=>done,
    error_id=>error_id
  );
  state_number := state_number + 10;
20:
  file.write(
    start:=FALSE,
    data_ptr:=ADR(message_queue.sGet),
    data_size:=TO_UDINT(LEN(message_queue.sGet)),
    done=>done,
    error_id=>error_id
  );
  
  IF done THEN
    state_number := 0;
	END_IF
END_CASE
END_METHOD

METHOD submit_event_message
VAR_IN_OUT
	ev: EventMessage;
END_VAR
IF ev.level >= level THEN
  message_queue.bLog := FALSE;
  message_queue.sPrefix := 'CSVLogger::';
  create_row(ev);
  message_queue.sPut := formatted_output.str;
  message_queue.AddTail();
END_IF
END_METHOD

END_FUNCTION_BLOCK

// ---- Utils/FB_FrameFifo.TcPOU
(* Tx/Rx (string data) fifo control function block *)
FUNCTION_BLOCK FB_FrameFifo
VAR_INPUT
	bLog		: BOOL			:= FALSE;(* TRUE => Enable log message output, FALSE => Disable *)
	sPrefix		: STRING		:= 'Unknown::';(* Log message description string (allows the identification of log message source) *)
	sPut		: T_MaxString 	:= ''; (* String message to add (write) to the fifo *)
END_VAR
VAR_OUTPUT
	bOk			: BOOL; 	 	(* TRUE = New entry added or removed succesfully, FALSE = Fifo overflow or fifo empty *)
	sGet		: T_MaxString 	:= '';(* String message removed (read) from fifo *)
	nCount		: UDINT			:= 0;(* Number of fifo entries *)
	cbFree		: UDINT 		:= 0;(* Free buffer space *)
END_VAR
VAR
	fbBuffer 	: FB_StringRingBuffer := (bOverwrite := FALSE);(* Basic (lower level) string buffer control function block *)
	buffer		: ARRAY[-3..Properties.CSV_BUFFER_SIZE] OF BYTE;(* Internal buffer memory *)
END_VAR

;

ACTION AddTail:
(* Adds new fifo entry *)
fbBuffer.A_AddTail( pBuffer:= ADR(buffer), cbBuffer:= SIZEOF(buffer),
					putValue:= sPut, bOk=>bOk, nCount=>nCount );
IF bOk THEN
	cbFree := Properties.CSV_BUFFER_SIZE - fbBuffer.cbSize;(* Calculate the free buffer space *)
	IF bLog THEN(* Log message *)
		ADSLOGSTR( ADSLOG_MSGTYPE_HINT OR ADSLOG_MSGTYPE_LOG, CONCAT( sPrefix, '<="%s"' ), sPut );
	END_IF
END_IF
END_ACTION

ACTION Clear:
(* Resets fifo = clears all data *)
fbBuffer.A_Reset( pBuffer:= ADR(buffer), cbBuffer:= SIZEOF(buffer),
				bOk=>bOk, getValue=>sGet, nCount=>nCount );
cbFree := Properties.CSV_BUFFER_SIZE;(* Free buffer size *)
END_ACTION

ACTION RemoveHead:
(* Removes oldest fifo entry *)
fbBuffer.A_RemoveHead( pBuffer:= ADR(buffer), cbBuffer:= SIZEOF(buffer),
						bOk=>bOk, getValue=>sGet, nCount=>nCount );
IF bOk THEN
	cbFree := Properties.CSV_BUFFER_SIZE - fbBuffer.cbSize;(* Calculate the free buffer space *)
END_IF
END_ACTION

END_FUNCTION_BLOCK

// ---- Utils/TIMESTRUCT_TO_DATESTR.TcPOU
FUNCTION TIMESTRUCT_TO_DATESTR
VAR_INPUT
  ts: TIMESTRUCT;
END_VAR
VAR_IN_OUT
  outputstr: STRING(255);
END_VAR
VAR
  format_string: FB_FormatString;
END_VAR

format_string(
  sFormat:='%d-%2d-%2d',
  arg1:=F_WORD(ts.wYear),
  arg2:=F_WORD(ts.wMonth),
  arg3:=F_WORD(ts.wDay),
  sOut=>outputstr);

END_FUNCTION

// ---- Logger/MemoryLogger.TcPOU
FUNCTION_BLOCK MemoryLogger IMPLEMENTS EventLogger
VAR_INPUT
END_VAR
VAR_OUTPUT
END_VAR
VAR
  event_history: ARRAY[1..Properties.MEMORY_LOGGER_NUM_EVENTS_HISTORY] OF EventMessageHMI;
  hmi_events: ARRAY[1..Properties.MEMORY_LOGGER_NUM_EVENTS_HMI] OF EventMessageHMI;
  _level: EventLevel;
  _hmi_level: EventLevel;
  act_time: TIMESTRUCT;
  act_time_str: STRING(255);
  format_string: FB_FormatString;
  _datetime_format: STRING(255) := '%4.0f-%02.0f-%02.0f %02.0f:%02.0f:%02.0f.%03.0f';
END_VAR

METHOD clear_event_message
VAR_INPUT
  id: INT;
END_VAR
// nothing to do here
END_METHOD

PROPERTY PUBLIC datetime_format : STRING(255)
GET
datetime_format := _datetime_format;
END_GET
SET
_datetime_format := datetime_format;
END_SET
END_PROPERTY

PROPERTY hmi_level : EventLevel
GET
hmi_level := _hmi_level;
END_GET
SET
_hmi_level := hmi_level;
END_SET
END_PROPERTY

PROPERTY PUBLIC level : EventLevel
GET
level := _level;
END_GET
SET
_level := level;
END_SET
END_PROPERTY

METHOD run
VAR_INPUT
	act_time	: Tc2_Utilities.TIMESTRUCT;
END_VAR
VAR_INST
  year: REAL;
  month: REAL;
  day: REAL;
  hour: REAL;
  minute: REAL;
  second: REAL;
  millisecond: REAL;
END_VAR
VAR
  i: INT;
  j: INT;
  empty_message: EventMessageHMI;
END_VAR
THIS^.act_time := act_time;
// ugly hack. have to convert numbers to real because the format specification
// only allows leading zeros on types f, e and s
year := TO_REAL(act_time.wYear);
month := TO_REAL(act_time.wMonth);
day := TO_REAL(act_time.wDay);
hour := TO_REAL(act_time.wHour);
minute := TO_REAL(act_time.wMinute);
second := TO_REAL(act_time.wSecond);
millisecond := TO_REAL(act_time.wMilliseconds);
format_string(
  sFormat:=datetime_format,
  arg1:=F_REAL(year),
  arg2:=F_REAL(month),
  arg3:=F_REAL(day),
  arg4:=F_REAL(hour),
  arg5:=F_REAL(minute),
  arg6:=F_REAL(second),
  arg7:=F_REAL(millisecond),
  sOut=>act_time_str);

j := 1;
FOR i:=1 TO Properties.MEMORY_LOGGER_NUM_EVENTS_HISTORY DO
  IF event_history[i].level >= hmi_level THEN
    hmi_events[j] := event_history[i];
    j := j + 1;
	END_IF
  IF j > Properties.MEMORY_LOGGER_NUM_EVENTS_HMI THEN
    EXIT;
	END_IF
END_FOR
WHILE j <= Properties.MEMORY_LOGGER_NUM_EVENTS_HMI DO
  hmi_events[j] := empty_message;
  j := j + 1;
END_WHILE
END_METHOD

METHOD submit_event_message
VAR_IN_OUT
	ev: EventMessage;
END_VAR
VAR_INST
  ev_hmi: EventMessageHMI;
END_VAR
IF ev.level >= level THEN
  ev_hmi.id := ev.id;
  ev_hmi.level := ev.level;
  ev_hmi.message := ev.message.str;
  ev_hmi.path := ev.path.str;
  ev_hmi.timestamp := act_time_str;
  put_new_data_at_start(SIZEOF(ev_hmi), ADR(ev_hmi), SIZEOF(event_history), ADR(event_history));
END_IF
END_METHOD

END_FUNCTION_BLOCK

// ---- Logger/AlarmViewLogger.TcPOU
FUNCTION_BLOCK AlarmViewLogger IMPLEMENTS EventLogger
VAR_INPUT
END_VAR
VAR_OUTPUT
END_VAR
VAR
  events: ARRAY[1..Properties.ALARM_VIEW_NUM_EVENTS] OF EventMessageHMI;
  empty_message: EventMessageHMI;
  _level: EventLevel;
  act_time: TIMESTRUCT;
  act_time_str: STRING(255);
  format_string: FB_FormatString;
  _datetime_format: STRING(255) := '%4.0f-%02.0f-%02.0f %02.0f:%02.0f:%02.0f.%03.0f';
END_VAR

METHOD clear_event_message
VAR_INPUT
	id: INT;
END_VAR
VAR
  index: INT;
  filldata: EventMessageHMI;
END_VAR
IF event_in_table(id:=id) THEN
  index := event_index(id:=id);
  
  remove_field_from_array(
    index_to_remove:=index,
    size_filldata:=SIZEOF(filldata),
    adr_filldata:=ADR(filldata),
    size_memory_buffer:=SIZEOF(events),
    adr_memory_buffer:=ADR(events));
END_IF
END_METHOD

PROPERTY PUBLIC datetime_format : STRING(255)
GET
datetime_format := _datetime_format;
END_GET
SET
_datetime_format := datetime_format;
END_SET
END_PROPERTY

METHOD PRIVATE event_in_table : BOOL
VAR_INPUT
  id: INT;
END_VAR
event_in_table := event_index(id) > 0;
END_METHOD

METHOD PRIVATE event_index : INT
VAR_INPUT
  id: INT;
END_VAR
VAR
  i: INT;
END_VAR
FOR i:=1 TO Properties.ALARM_VIEW_NUM_EVENTS DO
  // there are no gaps between events, so it is safe to assume
  // that the first empty event is the end
  IF events[i].id = 0 THEN
    EXIT;
	END_IF
  
  IF events[i].id := id THEN
    event_index := i;
    EXIT;
	END_IF
END_FOR
END_METHOD

PROPERTY PUBLIC level : EventLevel
GET
level := _level;
END_GET
SET
_level := level;
END_SET
END_PROPERTY

METHOD PUBLIC reset
VAR_INPUT
  execute: BOOL;
END_VAR
VAR
  i: INT;
END_VAR
VAR_INST
  r_execute: R_TRIG;
END_VAR
r_execute(CLK:=execute);
IF r_execute.Q THEN
  logging.reset_events_and_messages();
  FOR i:=1 TO Properties.ALARM_VIEW_NUM_EVENTS DO
    events[i] := empty_message;
	END_FOR
END_IF
END_METHOD

METHOD run
VAR_INPUT
	act_time	: Tc2_Utilities.TIMESTRUCT;
END_VAR
VAR_INST
  year: REAL;
  month: REAL;
  day: REAL;
  hour: REAL;
  minute: REAL;
  second: REAL;
  millisecond: REAL;
END_VAR
VAR
END_VAR
THIS^.act_time := act_time;
// ugly hack. have to convert numbers to real because the format specification
// only allows leading zeros on types f, e and s
year := TO_REAL(act_time.wYear);
month := TO_REAL(act_time.wMonth);
day := TO_REAL(act_time.wDay);
hour := TO_REAL(act_time.wHour);
minute := TO_REAL(act_time.wMinute);
second := TO_REAL(act_time.wSecond);
millisecond := TO_REAL(act_time.wMilliseconds);
format_string(
  sFormat:=datetime_format,
  arg1:=F_REAL(year),
  arg2:=F_REAL(month),
  arg3:=F_REAL(day),
  arg4:=F_REAL(hour),
  arg5:=F_REAL(minute),
  arg6:=F_REAL(second),
  arg7:=F_REAL(millisecond),
  sOut=>act_time_str);
END_METHOD

METHOD submit_event_message
VAR_IN_OUT
	ev: EventMessage;
END_VAR
VAR_INST
  ev_hmi: EventMessageHMI;
END_VAR
IF ev.level >= level THEN
  ev_hmi.id := ev.id;
  ev_hmi.level := ev.level;
  ev_hmi.message := ev.message.str;
  ev_hmi.path := ev.path.str;
  ev_hmi.timestamp := act_time_str;
  put_new_data_at_start(SIZEOF(ev_hmi), ADR(ev_hmi), SIZEOF(events), ADR(events));
END_IF
END_METHOD

END_FUNCTION_BLOCK

// ---- Tests/Event/TestEvent.TcPOU
FUNCTION_BLOCK TestEvent EXTENDS TcUnit.FB_TestSuite
VAR_INPUT
END_VAR
VAR_OUTPUT
END_VAR
VAR
END_VAR

create_event();
after_initialisation_alarm_is_not_raised();
after_raising_an_alarm_the_alarm_is_raised();
clear_alarm();
add_multiple_events();
raise_and_clear_multiple_alarms();

METHOD add_multiple_events
VAR_INST
  sut: MultipleEventTestsystem;
END_VAR
TEST('Add multiple events');

sut.event1.alarm();
sut.event2.warning();
sut.event3.alarm();
AssertTrue(sut.event1.alarm_raised, 'Event 1');
AssertFalse(sut.event2.alarm_raised, 'Event 2');
AssertTrue(sut.event3.alarm_raised, 'Event 3');

TEST_FINISHED();
END_METHOD

METHOD after_initialisation_alarm_is_not_raised
VAR_INPUT
END_VAR
VAR_INST
  sut: EventTestsystem;
END_VAR
TEST('Alarm is not raised after initialisation');

AssertFalse(sut.event.alarm_raised, '');

TEST_FINISHED();
END_METHOD

METHOD after_raising_an_alarm_the_alarm_is_raised
VAR_INPUT
END_VAR
VAR_INST
  sut: EventTestsystem;
END_VAR
TEST('After raising an alarm the alarm is raised');

sut.event.alarm();
AssertTrue(sut.event.alarm_raised, '');

TEST_FINISHED();
END_METHOD

METHOD clear_alarm
VAR_INPUT
END_VAR
VAR_INST
  sut: EventTestsystem;
END_VAR
TEST('Clear alarm');

sut.event.alarm();
sut.event.clear_alarm();
AssertFalse(sut.event.alarm_raised, '');

TEST_FINISHED();
END_METHOD

METHOD create_event
VAR_INPUT
END_VAR
VAR_INST
  sut: EventTestsystem;
END_VAR
TEST('Create event');

sut.event.message := 'Test';
AssertEquals_STRING('Test', sut.event.message, 'Event not properly created');

TEST_FINISHED();
END_METHOD

METHOD raise_and_clear_multiple_alarms
VAR_INST
  sut: MultipleEventTestsystem;
END_VAR
TEST('Raise and clear multiple alarms');

sut.event1.alarm();
sut.event2.alarm();
sut.event3.alarm();
sut.event1.clear_alarm();
sut.event3.clear_alarm();
AssertFalse(sut.event1.alarm_raised, 'Event 1');
AssertTrue(sut.event2.alarm_raised, 'Event 2');
AssertFalse(sut.event3.alarm_raised, 'Event 3');

TEST_FINISHED();
END_METHOD

END_FUNCTION_BLOCK

// ---- Tests/Logger/TestADSLogger.TcPOU
FUNCTION_BLOCK TestADSLogger EXTENDS TcUnit.FB_TestSuite
VAR_INPUT
END_VAR
VAR_OUTPUT
END_VAR
VAR
END_VAR

submit_info();
submit_warning();
submit_error();
submit_alarm();
change_default_level_to_warning_and_submit_info();
change_default_level_to_warning_and_submit_error();
create_event_with_a_parameter();
create_runner_message_with_a_parameter();
do_not_output_the_same_message_multiple_cycles_after_each_other();

METHOD change_default_level_to_warning_and_submit_error
VAR_INPUT
END_VAR
VAR_INST
  sut: ADSLoggerTestsystem;
END_VAR
VAR
  cut_output: STRING;
END_VAR
TEST('Change default level to warning and submit error');

sut.logging.add_logger(sut.logger);
sut.logger.level := EventLevel.WARNING;
sut.event.message := 'Default level warning';
sut.event.error();
cut_output := RIGHT(sut.logger.formatted_output.str, 31);

AssertEquals_DWORD(ADSLOG_MSGTYPE_ERROR, sut.logger.mask, '');
AssertEquals_STRING(' | ERROR: Default level warning', cut_output, '');

TEST_FINISHED();
END_METHOD

METHOD change_default_level_to_warning_and_submit_info
VAR_INPUT
END_VAR
VAR_INST
  sut: ADSLoggerTestsystem;
END_VAR
TEST('Change default level to warning and submit info');

sut.logging.add_logger(sut.logger);
sut.logger.level := EventLevel.WARNING;
sut.event.message := 'Default level warning';
sut.event.info();

AssertEquals_DWORD(0, sut.logger.mask, '');

TEST_FINISHED();
END_METHOD

METHOD create_event_with_a_parameter
VAR_INST
  sut: ADSLoggerTestsystem;
END_VAR
VAR
  parameter: INT;
  cut_output: STRING;
END_VAR
TEST('Create event with a parameter');

sut.logging.add_logger(sut.logger);
sut.event.message := 'Test %d';
parameter := 123;
sut.event.parameter := F_INT(parameter);
sut.event.error();
cut_output := RIGHT(sut.logger.formatted_output.str, 18);

AssertEquals_DWORD(ADSLOG_MSGTYPE_ERROR, sut.logger.mask, '');
AssertEquals_STRING(' | ERROR: Test 123', cut_output, '');

TEST_FINISHED();
END_METHOD

METHOD create_runner_message_with_a_parameter
VAR_INST
  sut: ADSLoggerTestsystem;
END_VAR
VAR
  parameter: REAL;
  cut_output: STRING;
END_VAR
TEST('Create runner message with a parameter');

sut.logging.add_logger(sut.logger);
parameter := 3.14;
sut.logging.parameter := F_REAL(parameter);
sut.logging.warning(message:='Test %1.2f');
cut_output := RIGHT(sut.logger.formatted_output.str, 21);

AssertEquals_STRING(' | WARNING: Test 3.14', cut_output, '');

TEST_FINISHED();
END_METHOD

METHOD do_not_output_the_same_message_multiple_cycles_after_each_other
VAR_INPUT
END_VAR
VAR_INST
  sut: ADSLoggerTestsystem;
  state_counter: INT;
END_VAR
VAR
  cut_output: STRING;
END_VAR
TEST('Do not output the same message multiple cycles after each other');

sut.logging.add_logger(sut.logger);
sut.logging.run();

CASE state_counter OF
0:
  sut.logging.error(message:='Alarm');
  sut.logging.error(message:='Error');
  
  cut_output := RIGHT(sut.logger.formatted_output.str, 15);
  
  AssertEquals_DWORD(ADSLOG_MSGTYPE_ERROR, sut.logger.mask, '');
  AssertEquals_STRING(' | ERROR: Error', cut_output, '');
  
  state_counter := state_counter + 10;
10:
  // do not output this message
  sut.logging.error(message:='Alarm');
  
  cut_output := RIGHT(sut.logger.formatted_output.str, 15);
  
  AssertEquals_STRING(' | ERROR: Error', cut_output, '');
  state_counter := state_counter + 10;
20:
  // do not output this message
  sut.logging.error(message:='Alarm');
  
  cut_output := RIGHT(sut.logger.formatted_output.str, 15);
  
  AssertEquals_STRING(' | ERROR: Error', cut_output, '');
  state_counter := state_counter + 10;
30:
  // do not output this message
  sut.logging.error(message:='Alarm');
  
  cut_output := RIGHT(sut.logger.formatted_output.str, 15);
  
  AssertEquals_STRING(' | ERROR: Error', cut_output, '');
  
  TEST_FINISHED();
END_CASE
END_METHOD

METHOD submit_alarm
VAR_INPUT
END_VAR
VAR_INST
  sut: ADSLoggerTestsystem;
END_VAR
VAR
  cut_output: STRING;
END_VAR
TEST('Submit alarm');

sut.logging.add_logger(sut.logger);
sut.event.message := 'Alarm';
sut.event.alarm();
cut_output := RIGHT(sut.logger.formatted_output.str, 15);

AssertEquals_DWORD(ADSLOG_MSGTYPE_ERROR, sut.logger.mask, '');
AssertEquals_STRING(' | ALARM: Alarm', cut_output, '');

TEST_FINISHED();
END_METHOD

METHOD submit_error
VAR_INPUT
END_VAR
VAR_INST
  sut: ADSLoggerTestsystem;
END_VAR
VAR
  cut_output: STRING;
END_VAR
TEST('Submit error');

sut.logging.add_logger(sut.logger);
sut.event.message := 'Error';
sut.event.error();
cut_output := RIGHT(sut.logger.formatted_output.str, 15);

AssertEquals_DWORD(ADSLOG_MSGTYPE_ERROR, sut.logger.mask, '');
AssertEquals_STRING(' | ERROR: Error', cut_output, '');

TEST_FINISHED();
END_METHOD

METHOD submit_info
VAR_INPUT
END_VAR
VAR_INST
  sut: ADSLoggerTestsystem;
END_VAR
VAR
  cut_output: STRING;
END_VAR
TEST('Submit info');

sut.logging.add_logger(sut.logger);
sut.event.message := 'Info';
sut.event.info();
cut_output := RIGHT(sut.logger.formatted_output.str, 13);

AssertEquals_DWORD(ADSLOG_MSGTYPE_HINT, sut.logger.mask, '');
AssertEquals_STRING(' | INFO: Info', cut_output, '');

TEST_FINISHED();
END_METHOD

METHOD submit_warning
VAR_INPUT
END_VAR
VAR_INST
  sut: ADSLoggerTestsystem;
END_VAR
VAR
  cut_output: STRING;
END_VAR
TEST('Submit warning');

sut.logging.add_logger(sut.logger);
sut.event.message := 'Warning';
sut.event.warning();
cut_output := RIGHT(sut.logger.formatted_output.str, 19);

AssertEquals_DWORD(ADSLOG_MSGTYPE_WARN, sut.logger.mask, '');
AssertEquals_STRING(' | WARNING: Warning', cut_output, '');

TEST_FINISHED();
END_METHOD

END_FUNCTION_BLOCK

// ---- Tests/Logger/TestCSVLogger.TcPOU
FUNCTION_BLOCK TestCSVLogger EXTENDS TcUnit.FB_TestSuite
VAR_INPUT
END_VAR
VAR_OUTPUT
END_VAR
VAR
END_VAR

submit_alarm();

METHOD submit_alarm
VAR_INPUT
END_VAR
VAR_INST
  sut: CSVLoggerTestsystem;
  state_number: INT;
END_VAR
TEST('Submit alarm');

sut.logging.run();

CASE state_number OF
0:
  IF sut.logging.time_valid THEN
    state_number := state_number + 10;
	END_IF
10:
  sut.logger.path := 'C:\';
  sut.logging.add_logger(sut.logger);
  sut.event.message := 'Alarm';
  sut.event.alarm();
  state_number := state_number + 10;
20:
  IF sut.logger.state_number = 0 THEN
    TEST_FINISHED();
	END_IF
END_CASE
END_METHOD

END_FUNCTION_BLOCK

// ---- Tests/TEST_MAIN.TcPOU
PROGRAM TEST_MAIN
VAR
  test_event: TestEvent;
  test_ads_logger: TestADSLogger;
  test_csv_logger: TestCSVLogger;
  test_utils: TestUtils;
END_VAR

TcUnit.RUN();
TEST_STRING_CYCLE_TIME();

END_PROGRAM

// ---- Tests/Utils/TestUtils.TcPOU
FUNCTION_BLOCK TestUtils EXTENDS TcUnit.FB_TestSuite
VAR_INPUT
END_VAR
VAR_OUTPUT
END_VAR
VAR
END_VAR

test_remove_project_from_path();

METHOD test_remove_project_from_path
VAR_INST
  path: LString;
END_VAR
TEST('Test remove project from path');

path.str := 'project.project.MAIN.test';
path.remove_left_including_char('.', 2);

AssertEquals_STRING('MAIN.test', path.str, '');

TEST_FINISHED();
END_METHOD

END_FUNCTION_BLOCK

// ---- Tests/TEST_STRING_CYCLE_TIME.TcPOU
PROGRAM TEST_STRING_CYCLE_TIME
VAR
  format_string: FB_FormatString;
  i: INT;
  j: INT;
  teststr: ARRAY[1..8] OF STRING(255);
  testlstr: ARRAY[1..8] OF LString;
  testtime: TIMESTRUCT;
  
  tst: INT;
END_VAR

testlstr[1].str := 'aaabbsbsbskjldajkgdklafk1';
testlstr[2].str := 'aaabbsbsbskjldajkgdklafk1';
testlstr[3].str := 'aaabbsbsbskjldajkgdklafk1';
testlstr[4].str := 'aaabbsbsbskjldajkgdklafk1';
testlstr[5].str := 'aaabbsbsbskjldajkgdklafk1';
teststr[1] := 'aaabbsbsbskjldajkgdklafk1';
teststr[2] := 'aaabbsbsbskjldajkgdklafk1';
teststr[3] := 'aaabbsbsbskjldajkgdklafk1';
teststr[4] := 'aaabbsbsbskjldajkgdklafk1';
teststr[5] := 'aaabbsbsbskjldajkgdklafk1';
testlstr[6].str := TO_STRING(testtime.wYear);
testlstr[6].str := TO_STRING(testtime.wMonth);
testlstr[6].str := TO_STRING(testtime.wDay);
FOR i:=1 TO 1000 DO
  (*TIMESTRUCT_TO_DATESTR(
    ts:=testtime,
    outputstr:=teststr[6]);
  TIMESTRUCT_TO_TIMESTR(
    ts:=testtime,
    outputstr:=teststr[7]);*)
  
  testlstr[6].str := '';
  testlstr[6].append(lstr:=testlstr[1]);
  testlstr[6].append(lstr:=testlstr[2]);
  testlstr[6].append(lstr:=testlstr[3]);
  testlstr[6].append(lstr:=testlstr[4]);
  testlstr[6].append(lstr:=testlstr[5]);
  (*format_string(
    sFormat:='%s,%s,%s,%s,%s$R',
    arg1:=F_STRING(teststr[1]),
    arg2:=F_STRING(teststr[2]),
    arg3:=F_STRING(teststr[3]),
    arg4:=F_STRING(teststr[4]),
    arg5:=F_STRING(teststr[5]),
    sOut=>teststr[6]
  );*)
END_FOR

END_PROGRAM

// ---- Utils/TIMESTRUCT_TO_TIMESTR.TcPOU
FUNCTION TIMESTRUCT_TO_TIMESTR
VAR_INPUT
  ts: TIMESTRUCT;
END_VAR
VAR_IN_OUT
  outputstr: STRING(255);
END_VAR
VAR
  format_string: FB_FormatString;
END_VAR

format_string(
  sFormat:='%2dh %2dm %2ds %3dms',
  arg1:=F_WORD(ts.wHour),
  arg2:=F_WORD(ts.wMinute),
  arg3:=F_WORD(ts.wSecond),
  arg4:=F_WORD(ts.wMilliseconds),
  sOut=>outputstr);

END_FUNCTION

// ---- GlobalTextList.TcGTLO
TEXTLIST GlobalTextList
  159 = '%s'
  866 = 'Path: %s'
  767 = 'Pfad: %s'
  243 = 'Reset'
END_TEXTLIST

// ---- Visu/AlarmViewMulti.TcVIS
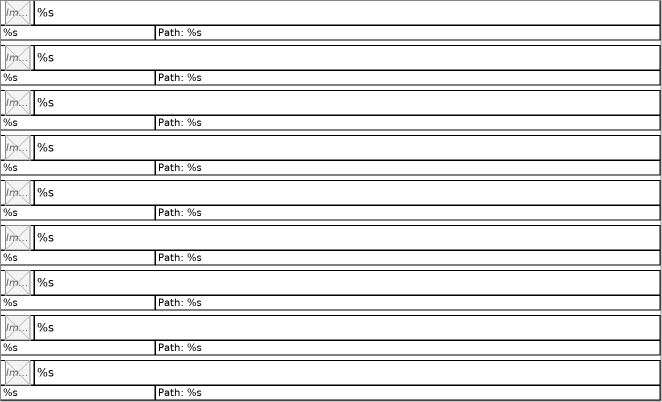
VISUALIZATION AlarmViewMulti  // 662x402
VAR_IN_OUT
	alarm_view: AlarmViewLogger;
END_VAR
    Frame (0,0 660x40), input disabled if: alarm_view.events[1].level = EventLevel.NONE
        shows AlarmViewSingle(event_message := alarm_view.events[1])
    Frame (0,45 660x40), input disabled if: alarm_view.events[2].level = EventLevel.NONE
        shows AlarmViewSingle(event_message := alarm_view.events[2])
    Frame (0,90 660x40), input disabled if: alarm_view.events[3].level = EventLevel.NONE
        shows AlarmViewSingle(event_message := alarm_view.events[3])
    Frame (0,135 660x40), input disabled if: alarm_view.events[4].level = EventLevel.NONE
        shows AlarmViewSingle(event_message := alarm_view.events[4])
    Frame (0,180 660x40), input disabled if: alarm_view.events[5].level = EventLevel.NONE
        shows AlarmViewSingle(event_message := alarm_view.events[5])
    Frame (0,225 660x40), input disabled if: alarm_view.events[6].level = EventLevel.NONE
        shows AlarmViewSingle(event_message := alarm_view.events[6])
    Frame (0,270 660x40), input disabled if: alarm_view.events[7].level = EventLevel.NONE
        shows AlarmViewSingle(event_message := alarm_view.events[7])
    Frame (0,315 660x40), input disabled if: alarm_view.events[8].level = EventLevel.NONE
        shows AlarmViewSingle(event_message := alarm_view.events[8])
    Frame (0,360 660x40), input disabled if: alarm_view.events[9].level = EventLevel.NONE
        shows AlarmViewSingle(event_message := alarm_view.events[9])
END_VISUALIZATION

// ---- Visu/AlarmViewSingle.TcVIS
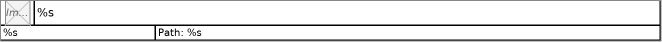
VISUALIZATION AlarmViewSingle  // 662x42
VAR_INPUT
	event_message: EventMessageHMI;
END_VAR
    Rectangle (0,25 155x15), "%s", text variable: event_message.timestamp
    Rectangle (0,0 34x25)
    Image (5,0 25x25)
        p84334746: GVL.IMAGE_ID[TO_INT(event_message.level)]
    Rectangle (34,0 626x25), "%s", text variable: event_message.message
    Rectangle (155,25 505x15), "Path: %s", text variable: event_message.path
END_VISUALIZATION

// ---- Visu/AlarmViewSingleWithReset.TcVIS
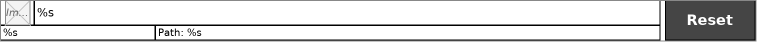
VISUALIZATION AlarmViewSingleWithReset  // 757x42
VAR_IN_OUT
  reset: BOOL;
END_VAR
VAR_INPUT
  event_message: EventMessageHMI;
  forward_visu: STRING;
END_VAR
    Frame (0,0 659x40)
        shows AlarmViewSingle(event_message := event_message)
        OnMouseClick: change screen: AssignExpression forward_visu
    Rectangle (665,0 90x40), "Reset"
        tap reset
END_VISUALIZATION
